FUNCTION_BLOCK Q_CtrlAudioSignal (* Command Control audio device ( Part 6 - F.10 ). *)
  (* Standard: ISO 11783-6; Description: Copyright (c) 2022 HR Agrartechnik GmbH This program and the accompanying materials are made available under the terms of the Eclipse Public License 2.0 which is available at https://www.eclipse.org/legal/epl-2.0/ SPDX-License-Identifier: EPL-2.0 see Description Tab *)
  (* Version 1.0, 2022-07-08, Franz Höpfinger, HR Agrartechnik GmbH *)
  PACKAGE isobus::UT::Q;
  IMPORT eclipse4diac::core::TypeHash;
  (* Documentation:
  Command Control audio device ( Part 6 - F.10 )
   This command can be used to control the audio on the VT.
   param[in] {u8NumOfRepit, uint8_t}
   Number of repetitions Range: 1 - 255
   param[in] {u16Frequency, uint16_t}
   Frequency
   param[in] {u16OnTimeMs, uint16_t}
   On time duration in ms
   param[in] {u16OffTimeMs, uint16_t}
   Off time duration in ms
   Return Values: 
   int16_t
    - VT_E_NO_ERR (0) - OK
   - VT_E_OVERFLOW (-6) - buffer overflow
   - VT_E_NOACT (-8) - Command not possible in current state
   - VT_E_NO_INSTANCE (-21) - No VT client available
   - VT_E_ISO_INSTANCE_INVALID (-129) - Identifier for instance (connection) invalid
   - VT_E_HANDLE_INVALID (-128) - ErrorCause: invalid Handle
   - VT_E_NOT_ALIVE (-130) - Identifier for instance valid, but VT Dead.
  *)
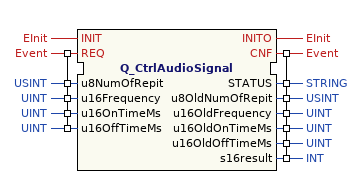
  EVENT_INPUT
    INIT : EInit; (* Service Initialization *)
    REQ WITH u8NumOfRepit, u16Frequency, u16OnTimeMs, u16OffTimeMs; (* Service Request *)
  END_EVENT
  EVENT_OUTPUT
    INITO : EInit; (* Initialization Confirm *)
    CNF WITH STATUS, u16OldOnTimeMs, u8OldNumOfRepit, u16OldFrequency, s16result, u16OldOffTimeMs; (* Confirmation of Requested Service *)
  END_EVENT
  VAR_INPUT
    u8NumOfRepit : USINT; (* Number of repetitions Range: 1 - 255 *)
    u16Frequency : UINT; (* Frequency *)
    u16OnTimeMs : UINT; (* On time duration in ms *)
    u16OffTimeMs : UINT; (* Off time duration in ms *)
  END_VAR
  VAR_OUTPUT
    STATUS : STRING; (* Service Status *)
    u8OldNumOfRepit : USINT; (* Old Number of repetitions Range: 1 - 255 *)
    u16OldFrequency : UINT; (* Old Frequency *)
    u16OldOnTimeMs : UINT; (* Old on time duration in ms *)
    u16OldOffTimeMs : UINT; (* Old off time duration in ms *)
    s16result : INT; (* retval see description *)
  END_VAR
END_FUNCTION_BLOCK
